(* Logix 5000 project; controller Comas_L4 vendor 1 type 14 code 193 rev 30.11; software revision 30.02; part 2 of 12 *)
(* tags used below, declared in another part *)
   Preposition_OK : BOOL;
(* Engage_Axe, continued *)

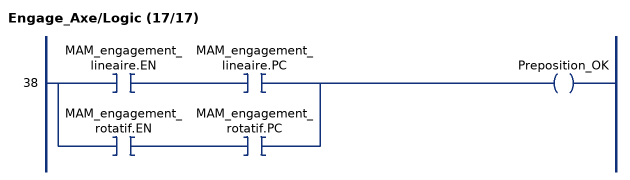
   38: [XIC(MAM_engagement_lineaire.EN) XIC(MAM_engagement_lineaire.PC) ,XIC(MAM_engagement_rotatif.EN) XIC(MAM_engagement_rotatif.PC) ]OTE(Preposition_OK);
END_ROUTINE
END_ADD_ON_INSTRUCTION

ADD_ON_INSTRUCTION Engage_Axe_Virtuel   (* revision 1.11 *)
// Revision note:
// v1.11: Modification Changement de Came en Synchro
// v1.10: Ajout des zones de changement de came
//            Mode Vnul optimisé
// v1.9: Correction Bug maitre à l'arret dans zone d'embrayage: (L16)
//    - Optimisation avec pending status
//    - Forward Only / Bi direc sur MAPC
//    - Command pos au lieu de actual pos sur MAPC
// v1.8: Lancement de came en mode Once (L17)
// v1.7: Degagemennt en position sur front (L8)
// v1.6: Retour cam engage Correct
// v1.5: Ajout modulo esclave
VAR_IN_OUT
   Axe : AXIS_VIRTUAL; {required}   // Axe esclave a controler
   Axe_Maitre : AXIS_VIRTUAL; {required}   // Axe maitre de la came
END_VAR
VAR_INPUT
   Activation : BOOL; {required}   // Activation puissance A Activer avant d'engager
   Engagement : BOOL; {required}   // Engagement de l'axe sur profil de came
   Maitre_V_Nul : BOOL; {required}   // Engagement avec Maitre vitesse nul (positionnement à l'arret)
   Engagement_Decalage : BOOL; {required}   // Activation du decalage en marche
   Degagement_en_pos : BOOL; {required}   // Attente position pour degagement
   Val_Vitesse : REAL; {required}   // Valeur de vitesse global de l'axe
   Val_Acc : REAL; {required}   // Valeur d accel gloable de laxe
   Val_Dec : REAL; {required}   // Valeur de decel
   Val_Jerk : REAL; {required}   // Valeur de jerk
   Val_Engagement : REAL; {required}   // Valeur Absolu d'engagement (0 ou 1 pour axe rotatif)
   Val_Degagement : REAL; {required}   // Valeur de degagement de l'axe (0 ou 1 pour axe rotatif)
   Val_Phase : REAL; {required}   // Valeur de Phase
   Val_Decalage : REAL; {required}   // Valeur de decalage (actif si bit d'activation a 1)
END_VAR
VAR_IN_OUT
   Came : CAM[100]; {required}   // Came modifiable a la volée (tableau de la came)
END_VAR
VAR_INPUT
   Longeur_Cam : DINT; {required}   // Longeur de la came (doit etre sup a 3)
   Modulo_Maitre : REAL; {required}   // Longeur du maitre pour calcul de la phase (modulo maitre)
   Mode_Rotatif : BOOL; {required}   // Activation mode rotatif (MAM type 2 au lieu de 0 pour le pre positionnement)
   Modulo_Esclave : DINT; {required}   // Utilise seulement pour engagement a vnul et rotatif (valeur du modulo de l'axe rotatif)
END_VAR
VAR_OUTPUT
   Axe_Engage : BOOL; {access Read Only, visible}   // Axe engage sur came
   Axe_Degage : BOOL; {access Read Only, visible}   // Axe Degage
   ER : BOOL; {access Read Only, visible}   // Erreur dans le module (retour des blocs fonction)
END_VAR
VAR_INPUT
   Num_Cam_Vnul : DINT;
   ModeCamOnce : BOOL; {required}   // Came en mode once (actif = 1)
   Top_Once : BOOL; {required}   // Top de lancement en mode once
END_VAR
VAR
   MAS_degagement : MOTION_INSTRUCTION;
   MAS_Engagement : MOTION_INSTRUCTION;
   MCCP_1 : MOTION_INSTRUCTION;
   Came_Prof_1 : CAM_PROFILE[20];
   MAPC_1 : MOTION_INSTRUCTION;
   Front : BOOL;
   Val_Phase_Sauve : REAL;
   Val_Phase_Modifie : REAL;
   MAM_Phase : MOTION_INSTRUCTION;
   Engagement_came : BOOL;
   MAM_decalage : MOTION_INSTRUCTION;
   MCCP_2 : MOTION_INSTRUCTION;
   MCCP_First : MOTION_INSTRUCTION;
   MAPC_First : MOTION_INSTRUCTION;
   Came_Prof_2 : CAM_PROFILE[20];
   Came_Prof_First : CAM_PROFILE[20];
   MAPC_2 : MOTION_INSTRUCTION;
   Top_Calage0 : BOOL;
   TEMP_0 : BOOL;
   TEMP_1 : BOOL;
   Top_Calage1 : BOOL;
   Axe_Active : BOOL;
   Num_Cam : DINT;
   Val_phase_modulo : REAL;
   Erreur_1 : BOOL;
   Erreur_2 : BOOL;
   MAS_degagement_enpos : MOTION_INSTRUCTION;
   DEGagement_En_Pos_ok : BOOL;
   Top_Calage2 : BOOL;
   TEMP_2 : BOOL;
   TEMP_3 : BOOL;
   Top_Calage3 : BOOL;
   Val_Engagement_plus : REAL;
   MAM_degagement_rotatif : MOTION_INSTRUCTION;
   MAM_degagement_lineaire : MOTION_INSTRUCTION;
   MAM_degagement_enpos_lineaire : MOTION_INSTRUCTION;
   MAM_degagement_enpos_rotatif : MOTION_INSTRUCTION;
   MAM_engagement_rotatif : MOTION_INSTRUCTION;
   MAM_engagement_lineaire : MOTION_INSTRUCTION;
   Degagement_en_pos_demande : BOOL;
   MAS_degagement_maitreVnul : MOTION_INSTRUCTION;
   Engagement_came_VNul : BOOL;
   MCCP_First_Vnul : MOTION_INSTRUCTION;
   MCSV_Slave_Value : REAL;
   MCSV_Slope_Value : REAL;
   MCSV_SlopeD_Value : REAL;
   MCSV : MOTION_INSTRUCTION;
   MAM_engagement_lineaire_vnul : MOTION_INSTRUCTION;
   MAM_engagement_rotatifvnul : MOTION_INSTRUCTION;
   Val_MAitre : REAL;
   MAPC_First_Vnul : MOTION_INSTRUCTION;
   Front_vnul : BOOL;
   Val_Phase_Modulo2 : REAL;
   MCCP_1_vnul : MOTION_INSTRUCTION;
   Came_Prof_1_vnul : CAM_PROFILE[20];
   MAPC_1_vnul : MOTION_INSTRUCTION;
   MCCP_2_vnul : MOTION_INSTRUCTION;
   Came_Prof_2_vnul : CAM_PROFILE[20];
   MAPC_2_vnul : MOTION_INSTRUCTION;
   TEMP_5 : BOOL;
   Top_Calage5 : BOOL;
   TEMP_6 : BOOL;
   Top_Calage6 : BOOL;
   Erreur_3 : BOOL;
   Erreur_4 : BOOL;
   Front200 : BOOL;
   Cam_Pending : BOOL;
   Tempo_degagement : TIMER;
   decalage_Vnul_Dem : REAL;
   decalage_Vnul_Dem_modulo : REAL;
   front_degagement : BOOL; {access None}
   modulo_div2 : REAL := 1.0; {access None}
   MCCP_First_Once : MOTION_INSTRUCTION; {access None}
   Came_Prof_First_Once : CAM_PROFILE[20]; {access None}
   MAPC_First_Once : MOTION_INSTRUCTION; {access None}
   Front_once : BOOL; {access None}
   Synchro_0 : BOOL; {access None}
   Synchro_1 : BOOL; {access None}
   Val_Engagement_plus_min : REAL; {access None}
   Synchro_vnul_0 : BOOL; {access None}
   Synchro_vnul_1 : BOOL; {access None}
END_VAR

ROUTINE Logic   (* ladder *)
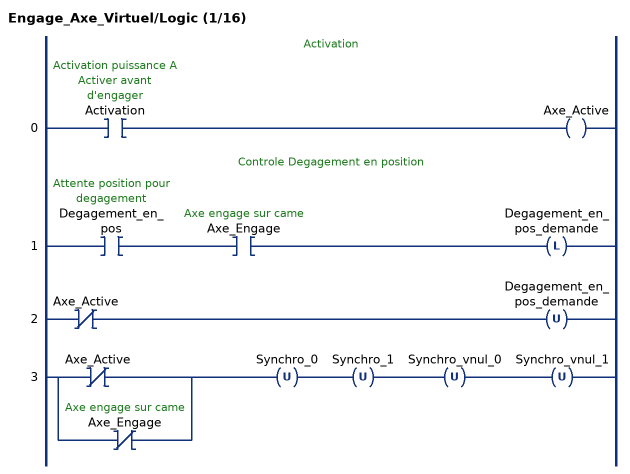
   // Activation
   0: XIC(Activation)OTE(Axe_Active);
   // Controle Degagement en position
   1: XIC(Degagement_en_pos)XIC(Axe_Engage)OTL(Degagement_en_pos_demande);
   2: XIO(Axe_Active)OTU(Degagement_en_pos_demande);
   3: [XIO(Axe_Active) ,XIO(Axe_Engage) ]OTU(Synchro_0)OTU(Synchro_1)OTU(Synchro_vnul_0)OTU(Synchro_vnul_1);
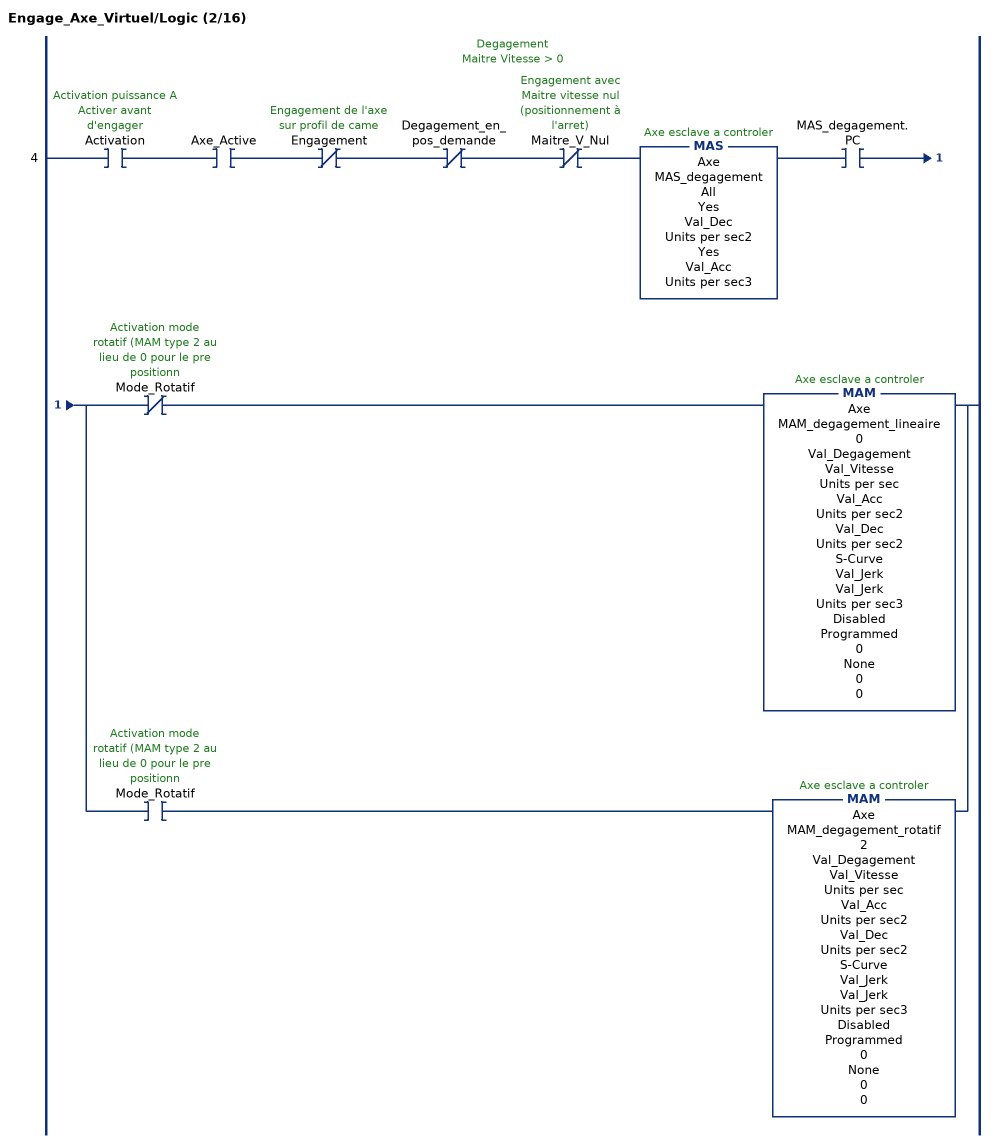
   // Degagement
   // Maitre Vitesse > 0
   4: XIC(Activation)XIC(Axe_Active)XIO(Engagement)XIO(Degagement_en_pos_demande)XIO(Maitre_V_Nul)MAS(Axe,MAS_degagement,All,Yes,Val_Dec,Units per sec2,Yes,Val_Acc,Units per sec3)XIC(MAS_degagement.PC)[XIO(Mode_Rotatif) MAM(Axe,MAM_degagement_lineaire,0,Val_Degagement,Val_Vitesse,Units per sec,Val_Acc,Units per sec2,Val_Dec,Units per sec2,S-Curve,Val_Jerk,Val_Jerk,Units per sec3,Disabled,Programmed,0,None,0,0) ,XIC(Mode_Rotatif) MAM(Axe,MAM_degagement_rotatif,2,Val_Degagement,Val_Vitesse,Units per sec,Val_Acc,Units per sec2,Val_Dec,Units per sec2,S-Curve,Val_Jerk,Val_Jerk,Units per sec3,Disabled,Programmed,0,None,0,0) ];
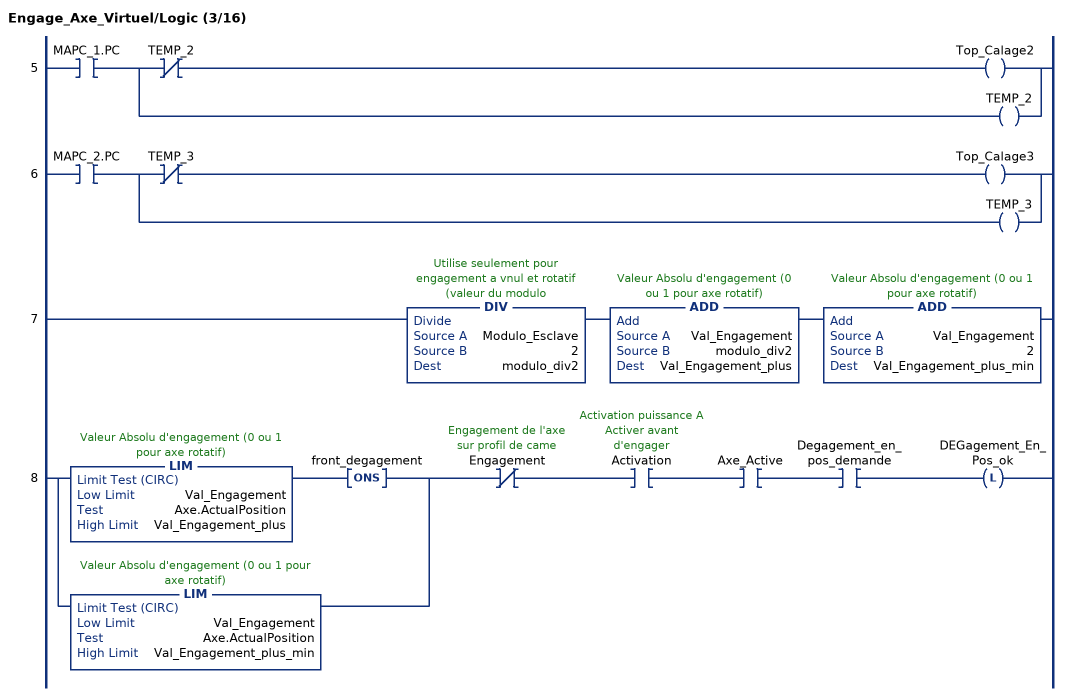
   5: XIC(MAPC_1.PC)[XIO(TEMP_2) OTE(Top_Calage2) ,OTE(TEMP_2) ];
   6: XIC(MAPC_2.PC)[XIO(TEMP_3) OTE(Top_Calage3) ,OTE(TEMP_3) ];
   7: DIV(Modulo_Esclave,2,modulo_div2)ADD(Val_Engagement,modulo_div2,Val_Engagement_plus)ADD(Val_Engagement,2,Val_Engagement_plus_min);
   8: [LIM(Val_Engagement,Axe.ActualPosition,Val_Engagement_plus) ONS(front_degagement) ,LIM(Val_Engagement,Axe.ActualPosition,Val_Engagement_plus_min) ]XIO(Engagement)XIC(Activation)XIC(Axe_Active)XIC(Degagement_en_pos_demande)OTL(DEGagement_En_Pos_ok);
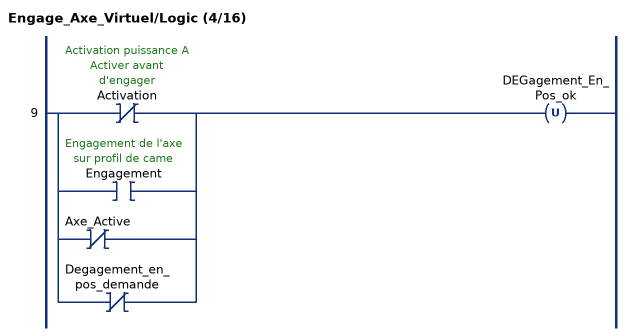
   9: [XIO(Activation) ,XIC(Engagement) ,XIO(Axe_Active) ,XIO(Degagement_en_pos_demande) ]OTU(DEGagement_En_Pos_ok);
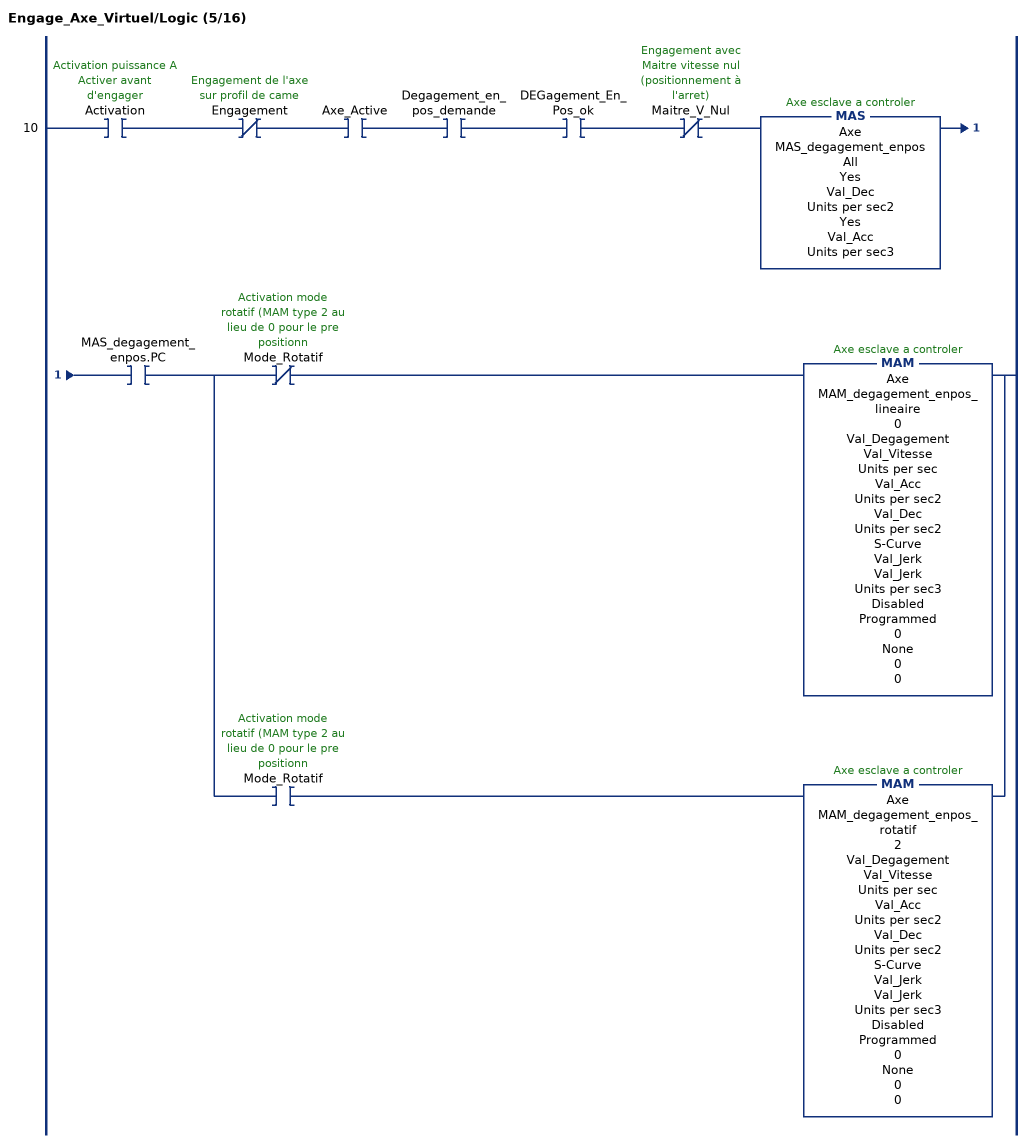
   10: XIC(Activation)XIO(Engagement)XIC(Axe_Active)XIC(Degagement_en_pos_demande)XIC(DEGagement_En_Pos_ok)XIO(Maitre_V_Nul)MAS(Axe,MAS_degagement_enpos,All,Yes,Val_Dec,Units per sec2,Yes,Val_Acc,Units per sec3)XIC(MAS_degagement_enpos.PC)[XIO(Mode_Rotatif) MAM(Axe,MAM_degagement_enpos_lineaire,0,Val_Degagement,Val_Vitesse,Units per sec,Val_Acc,Units per sec2,Val_Dec,Units per sec2,S-Curve,Val_Jerk,Val_Jerk,Units per sec3,Disabled,Programmed,0,None,0,0) ,XIC(Mode_Rotatif) MAM(Axe,MAM_degagement_enpos_rotatif,2,Val_Degagement,Val_Vitesse,Units per sec,Val_Acc,Units per sec2,Val_Dec,Units per sec2,S-Curve,Val_Jerk,Val_Jerk,Units per sec3,Disabled,Programmed,0,None,0,0) ];
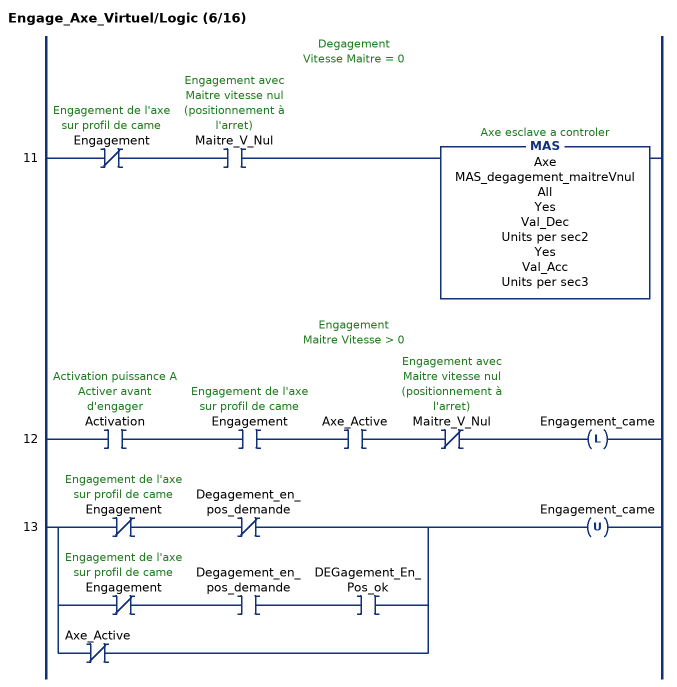
   // Degagement
   // Vitesse Maitre = 0
   11: XIO(Engagement)XIC(Maitre_V_Nul)MAS(Axe,MAS_degagement_maitreVnul,All,Yes,Val_Dec,Units per sec2,Yes,Val_Acc,Units per sec3);
   // Engagement
   // Maitre Vitesse > 0
   12: XIC(Activation)XIC(Engagement)XIC(Axe_Active)XIO(Maitre_V_Nul)OTL(Engagement_came);
   13: [XIO(Engagement) XIO(Degagement_en_pos_demande) ,XIO(Engagement) XIC(Degagement_en_pos_demande) XIC(DEGagement_En_Pos_ok) ,XIO(Axe_Active) ]OTU(Engagement_came);
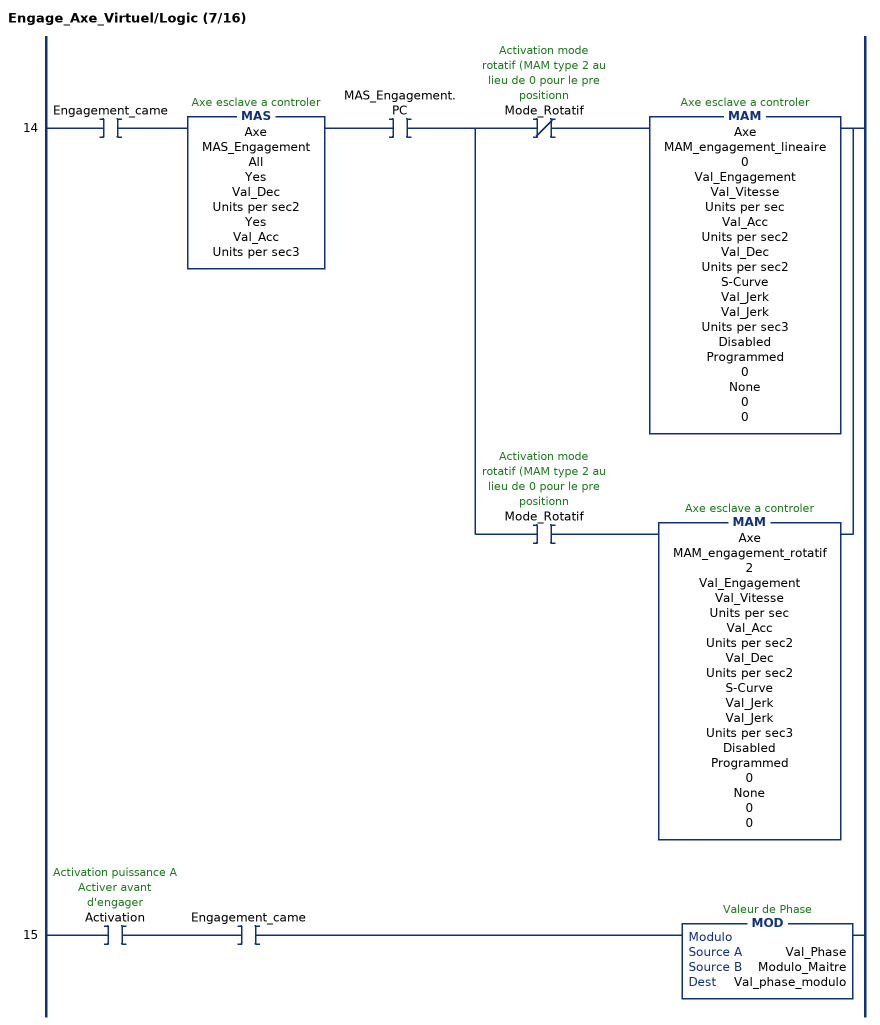
   14: XIC(Engagement_came)MAS(Axe,MAS_Engagement,All,Yes,Val_Dec,Units per sec2,Yes,Val_Acc,Units per sec3)XIC(MAS_Engagement.PC)[XIO(Mode_Rotatif) MAM(Axe,MAM_engagement_lineaire,0,Val_Engagement,Val_Vitesse,Units per sec,Val_Acc,Units per sec2,Val_Dec,Units per sec2,S-Curve,Val_Jerk,Val_Jerk,Units per sec3,Disabled,Programmed,0,None,0,0) ,XIC(Mode_Rotatif) MAM(Axe,MAM_engagement_rotatif,2,Val_Engagement,Val_Vitesse,Units per sec,Val_Acc,Units per sec2,Val_Dec,Units per sec2,S-Curve,Val_Jerk,Val_Jerk,Units per sec3,Disabled,Programmed,0,None,0,0) ];
   15: XIC(Activation)XIC(Engagement_came)MOD(Val_Phase,Modulo_Maitre,Val_phase_modulo);
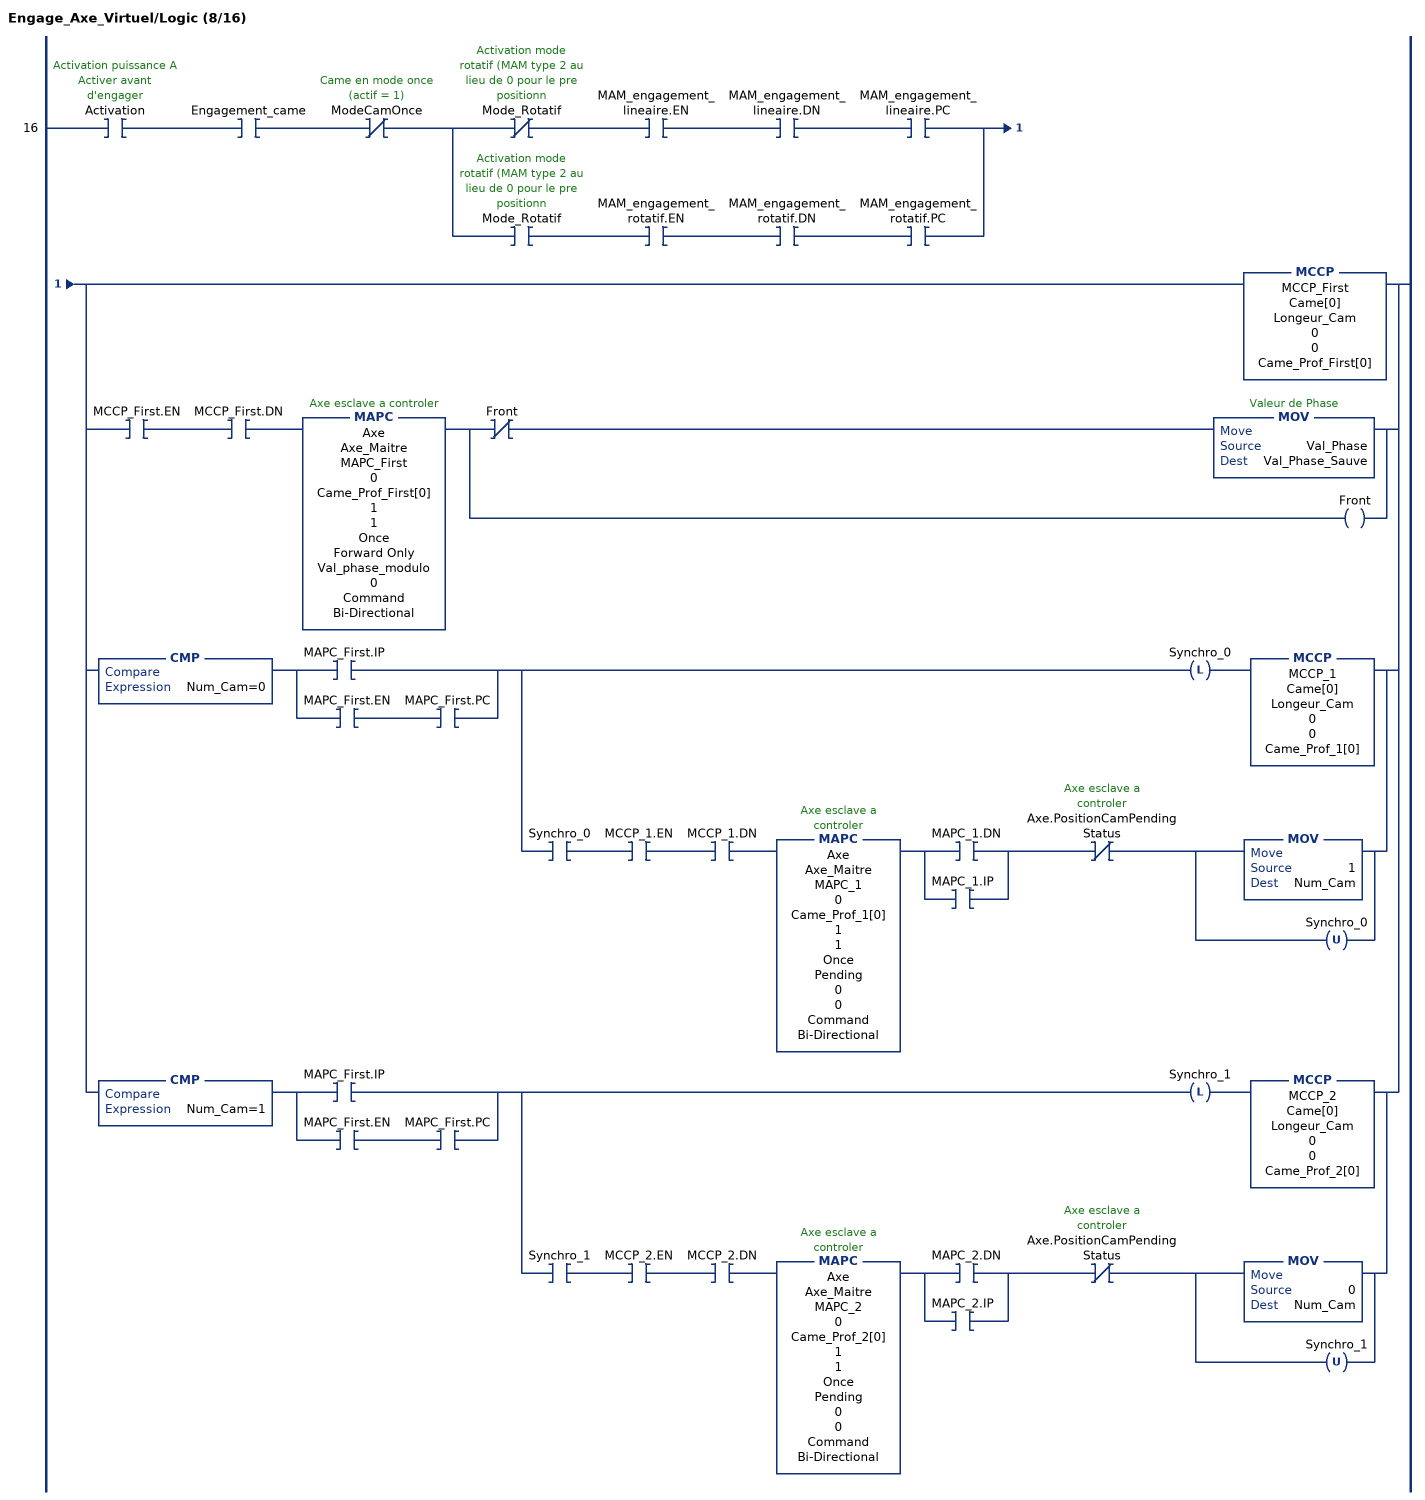
   16: XIC(Activation)XIC(Engagement_came)XIO(ModeCamOnce)[XIO(Mode_Rotatif) XIC(MAM_engagement_lineaire.EN) XIC(MAM_engagement_lineaire.DN) XIC(MAM_engagement_lineaire.PC) ,XIC(Mode_Rotatif) XIC(MAM_engagement_rotatif.EN) XIC(MAM_engagement_rotatif.DN) XIC(MAM_engagement_rotatif.PC) ][MCCP(MCCP_First,Came[0],Longeur_Cam,0,0,Came_Prof_First[0]) ,[XIC(MCCP_First.EN) XIC(MCCP_First.DN) MAPC(Axe,Axe_Maitre,MAPC_First,0,Came_Prof_First[0],1,1,Once,Forward Only,Val_phase_modulo,0,Command,Bi-Directional) [XIO(Front) MOV(Val_Phase,Val_Phase_Sauve) ,OTE(Front) ] ,CMP(Num_Cam=0) [XIC(MAPC_First.IP) ,XIC(MAPC_First.EN) XIC(MAPC_First.PC) ] [OTL(Synchro_0) MCCP(MCCP_1,Came[0],Longeur_Cam,0,0,Came_Prof_1[0]) ,XIC(Synchro_0) XIC(MCCP_1.EN) XIC(MCCP_1.DN) MAPC(Axe,Axe_Maitre,MAPC_1,0,Came_Prof_1[0],1,1,Once,Pending,0,0,Command,Bi-Directional) [XIC(MAPC_1.DN) ,XIC(MAPC_1.IP) ] XIO(Axe.PositionCamPendingStatus) [MOV(1,Num_Cam) ,OTU(Synchro_0) ] ] ,CMP(Num_Cam=1) [XIC(MAPC_First.IP) ,XIC(MAPC_First.EN) XIC(MAPC_First.PC) ] [OTL(Synchro_1) MCCP(MCCP_2,Came[0],Longeur_Cam,0,0,Came_Prof_2[0]) ,XIC(Synchro_1) XIC(MCCP_2.EN) XIC(MCCP_2.DN) MAPC(Axe,Axe_Maitre,MAPC_2,0,Came_Prof_2[0],1,1,Once,Pending,0,0,Command,Bi-Directional) [XIC(MAPC_2.DN) ,XIC(MAPC_2.IP) ] XIO(Axe.PositionCamPendingStatus) [MOV(0,Num_Cam) ,OTU(Synchro_1) ] ] ] ];
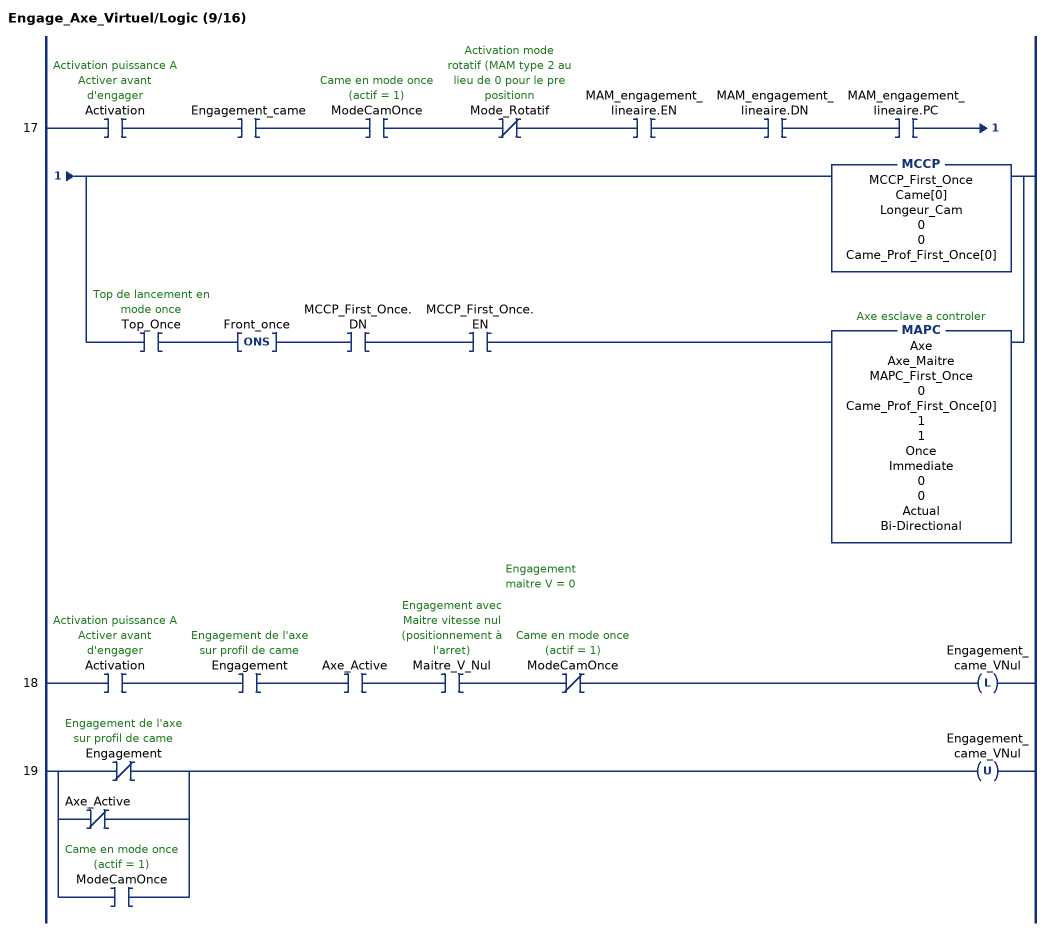
   17: XIC(Activation)XIC(Engagement_came)XIC(ModeCamOnce)XIO(Mode_Rotatif)XIC(MAM_engagement_lineaire.EN)XIC(MAM_engagement_lineaire.DN)XIC(MAM_engagement_lineaire.PC)[MCCP(MCCP_First_Once,Came[0],Longeur_Cam,0,0,Came_Prof_First_Once[0]) ,XIC(Top_Once) ONS(Front_once) XIC(MCCP_First_Once.DN) XIC(MCCP_First_Once.EN) MAPC(Axe,Axe_Maitre,MAPC_First_Once,0,Came_Prof_First_Once[0],1,1,Once,Immediate,0,0,Actual,Bi-Directional) ];
   // Engagement
   // maitre V = 0
   18: XIC(Activation)XIC(Engagement)XIC(Axe_Active)XIC(Maitre_V_Nul)XIO(ModeCamOnce)OTL(Engagement_came_VNul);
   19: [XIO(Engagement) ,XIO(Axe_Active) ,XIC(ModeCamOnce) ]OTU(Engagement_came_VNul);
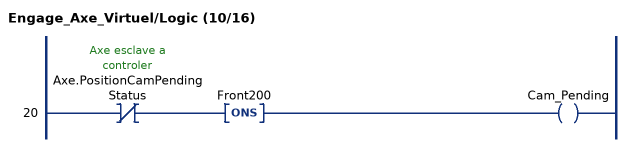
   20: XIO(Axe.PositionCamPendingStatus)ONS(Front200)OTE(Cam_Pending);
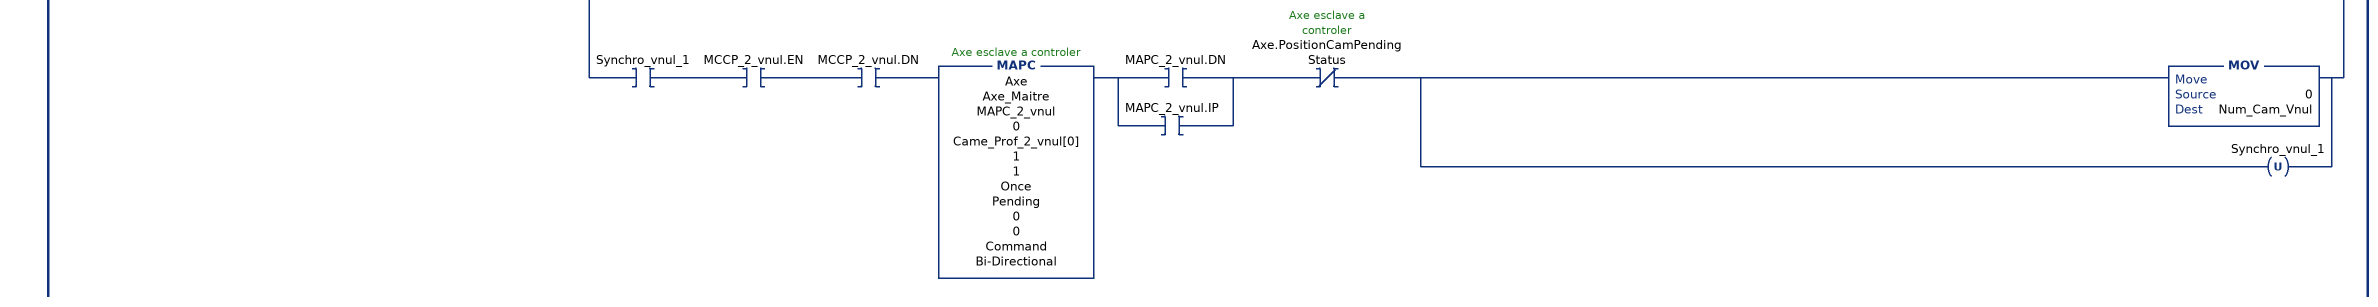
   21: XIC(Engagement_came_VNul)[MCCP(MCCP_First_Vnul,Came[0],Longeur_Cam,0,0,Came_Prof_First[0]) ,XIC(MCCP_First_Vnul.EN) XIC(MCCP_First_Vnul.DN) MOD(Val_Phase,Modulo_Maitre,Val_Phase_Modulo2) SUB(Axe_Maitre.CommandPosition,Val_Phase_Modulo2,Val_MAitre) ADD(Val_MAitre,Modulo_Maitre,Val_MAitre) MOD(Val_MAitre,Modulo_Maitre,Val_MAitre) MCSV(MCSV,Came_Prof_First[0],Val_MAitre,MCSV_Slave_Value,MCSV_Slope_Value,MCSV_SlopeD_Value) ADD(MCSV_Slave_Value,Val_Engagement,decalage_Vnul_Dem) MOD(decalage_Vnul_Dem,Modulo_Esclave,decalage_Vnul_Dem_modulo) XIC(MCSV.DN) [XIO(Mode_Rotatif) MAM(Axe,MAM_engagement_lineaire_vnul,0,decalage_Vnul_Dem,Val_Vitesse,Units per sec,Val_Acc,Units per sec2,Val_Dec,Units per sec2,S-Curve,Val_Jerk,Val_Jerk,Units per sec3,Disabled,Programmed,0,None,0,0) ,XIC(Mode_Rotatif) MAM(Axe,MAM_engagement_rotatifvnul,2,decalage_Vnul_Dem_modulo,Val_Vitesse,Units per sec,Val_Acc,Units per sec2,Val_Dec,Units per sec2,S-Curve,Val_Jerk,Val_Jerk,Units per sec3,Disabled,Programmed,0,None,0,0) ] ,XIC(MCCP_First_Vnul.EN) XIC(MCCP_First_Vnul.DN) MAPC(Axe,Axe_Maitre,MAPC_First_Vnul,0,Came_Prof_First[0],1,1,Once,Immediate,0,Val_MAitre,Command,Bi-Directional) [XIO(Front_vnul) MOV(Val_Phase,Val_Phase_Sauve) ,OTE(Front_vnul) ] ,CMP(Num_Cam_Vnul=0) [XIC(MAPC_First_Vnul.IP) ,XIC(MAPC_First_Vnul.EN) XIC(MAPC_First_Vnul.PC) ] [OTL(Synchro_vnul_0) MCCP(MCCP_1_vnul,Came[0],Longeur_Cam,0,0,Came_Prof_1_vnul[0]) ,XIC(Synchro_vnul_0) XIC(MCCP_1_vnul.EN) XIC(MCCP_1_vnul.DN) MAPC(Axe,Axe_Maitre,MAPC_1_vnul,0,Came_Prof_1_vnul[0],1,1,Once,Pending,0,0,Command,Bi-Directional) [XIC(MAPC_1_vnul.DN) ,XIC(MAPC_1_vnul.IP) ] XIO(Axe.PositionCamPendingStatus) [MOV(1,Num_Cam_Vnul) ,OTU(Synchro_vnul_0) ] ] ,CMP(Num_Cam_Vnul=1) [XIC(MAPC_First_Vnul.IP) ,XIC(MAPC_First_Vnul.EN) XIC(MAPC_First_Vnul.PC) ] [OTL(Synchro_vnul_1) MCCP(MCCP_2_vnul,Came[0],Longeur_Cam,0,0,Came_Prof_2_vnul[0]) ,XIC(Synchro_vnul_1) XIC(MCCP_2_vnul.EN) XIC(MCCP_2_vnul.DN) MAPC(Axe,Axe_Maitre,MAPC_2_vnul,0,Came_Prof_2_vnul[0],1,1,Once,Pending,0,0,Command,Bi-Directional) [XIC(MAPC_2_vnul.DN) ,XIC(MAPC_2_vnul.IP) ] XIO(Axe.PositionCamPendingStatus) [MOV(0,Num_Cam_Vnul) ,OTU(Synchro_vnul_1) ] ] ];
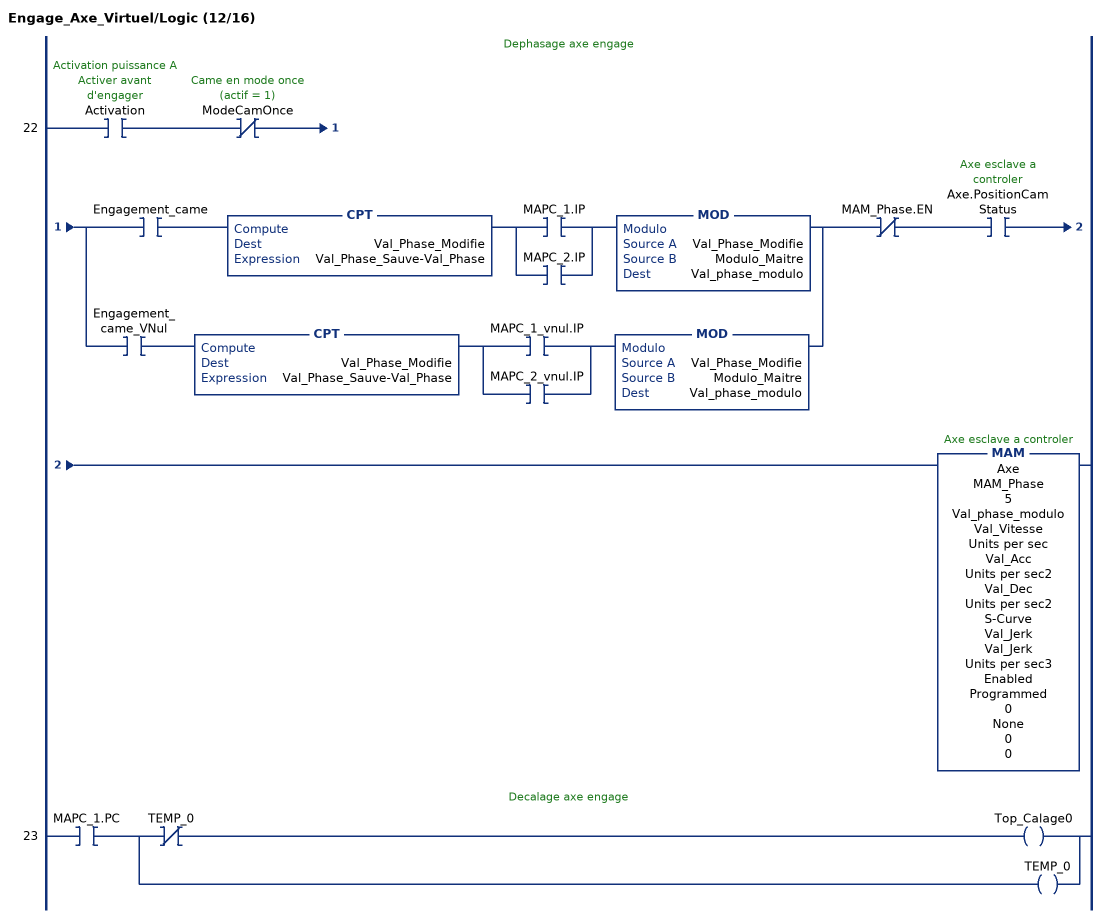
   // Dephasage axe engage
   22: XIC(Activation)XIO(ModeCamOnce)[XIC(Engagement_came) CPT(Val_Phase_Modifie,Val_Phase_Sauve-Val_Phase) [XIC(MAPC_1.IP) ,XIC(MAPC_2.IP) ] MOD(Val_Phase_Modifie,Modulo_Maitre,Val_phase_modulo) ,XIC(Engagement_came_VNul) CPT(Val_Phase_Modifie,Val_Phase_Sauve-Val_Phase) [XIC(MAPC_1_vnul.IP) ,XIC(MAPC_2_vnul.IP) ] MOD(Val_Phase_Modifie,Modulo_Maitre,Val_phase_modulo) ]XIO(MAM_Phase.EN)XIC(Axe.PositionCamStatus)MAM(Axe,MAM_Phase,5,Val_phase_modulo,Val_Vitesse,Units per sec,Val_Acc,Units per sec2,Val_Dec,Units per sec2,S-Curve,Val_Jerk,Val_Jerk,Units per sec3,Enabled,Programmed,0,None,0,0);
   // Decalage axe engage
   23: XIC(MAPC_1.PC)[XIO(TEMP_0) OTE(Top_Calage0) ,OTE(TEMP_0) ];
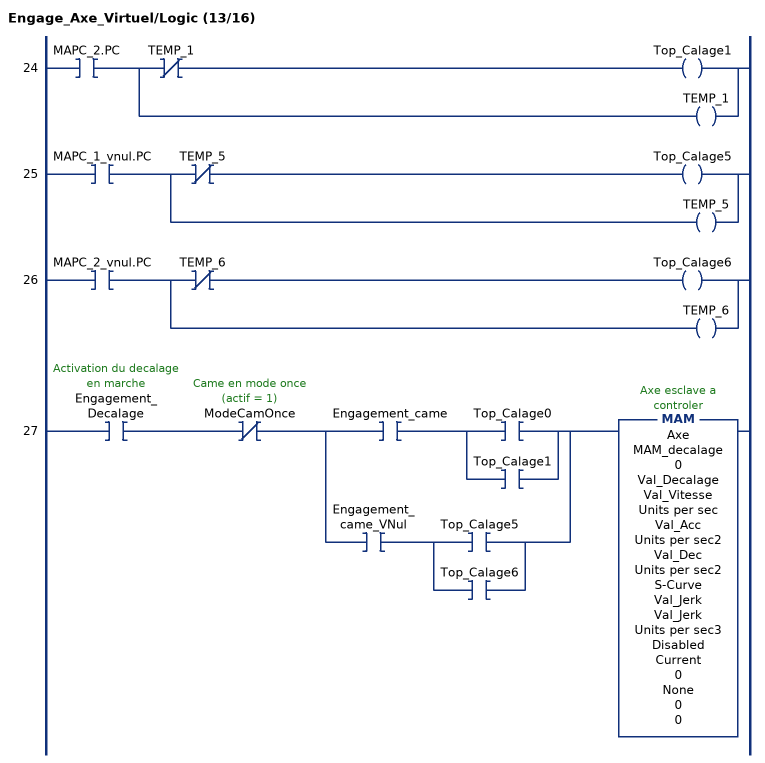
   24: XIC(MAPC_2.PC)[XIO(TEMP_1) OTE(Top_Calage1) ,OTE(TEMP_1) ];
   25: XIC(MAPC_1_vnul.PC)[XIO(TEMP_5) OTE(Top_Calage5) ,OTE(TEMP_5) ];
   26: XIC(MAPC_2_vnul.PC)[XIO(TEMP_6) OTE(Top_Calage6) ,OTE(TEMP_6) ];
   27: XIC(Engagement_Decalage)XIO(ModeCamOnce)[XIC(Engagement_came) [XIC(Top_Calage0) ,XIC(Top_Calage1) ] ,XIC(Engagement_came_VNul) [XIC(Top_Calage5) ,XIC(Top_Calage6) ] ]MAM(Axe,MAM_decalage,0,Val_Decalage,Val_Vitesse,Units per sec,Val_Acc,Units per sec2,Val_Dec,Units per sec2,S-Curve,Val_Jerk,Val_Jerk,Units per sec3,Disabled,Current,0,None,0,0);
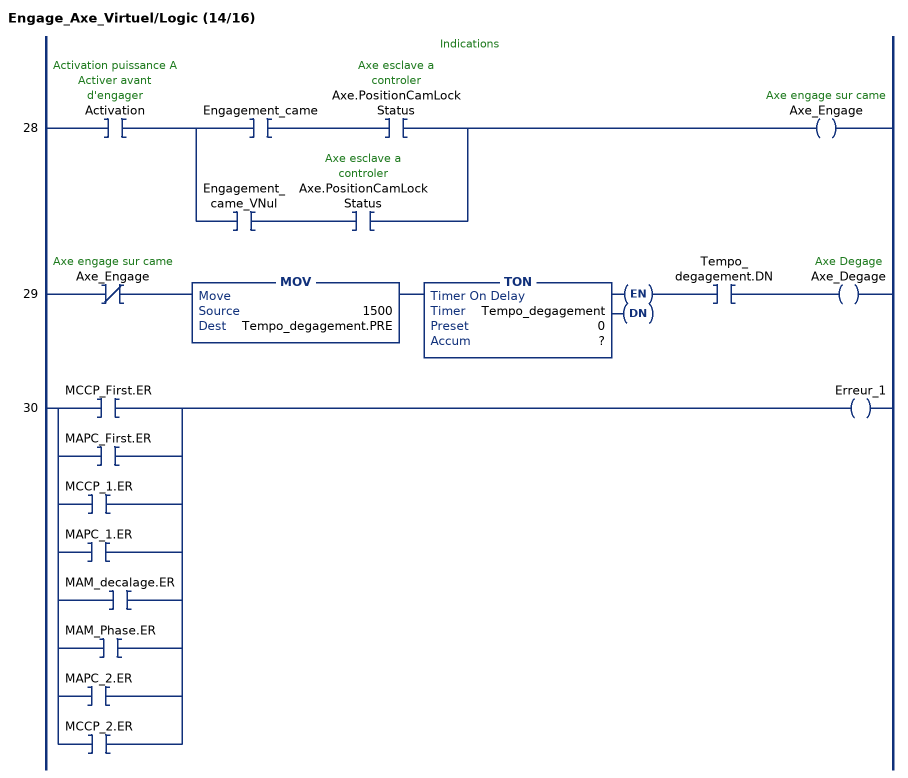
   // Indications
   28: XIC(Activation)[XIC(Engagement_came) XIC(Axe.PositionCamLockStatus) ,XIC(Engagement_came_VNul) XIC(Axe.PositionCamLockStatus) ]OTE(Axe_Engage);
   29: XIO(Axe_Engage)MOV(1500,Tempo_degagement.PRE)TON(Tempo_degagement,?,?)XIC(Tempo_degagement.DN)OTE(Axe_Degage);
   30: [XIC(MCCP_First.ER) ,XIC(MAPC_First.ER) ,XIC(MCCP_1.ER) ,XIC(MAPC_1.ER) ,XIC(MAM_decalage.ER) ,XIC(MAM_Phase.ER) ,XIC(MAPC_2.ER) ,XIC(MCCP_2.ER) ]OTE(Erreur_1);
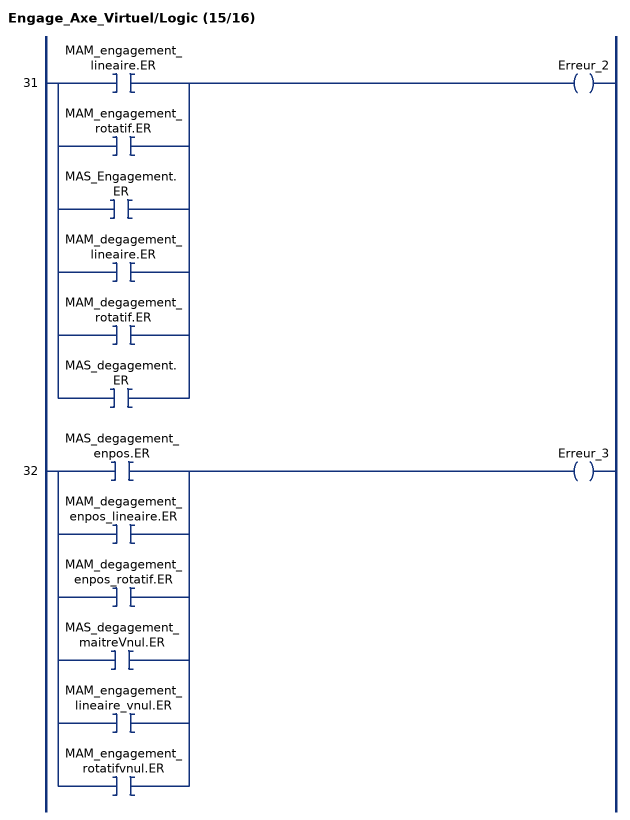
   31: [[XIC(MAM_engagement_lineaire.ER) ,XIC(MAM_engagement_rotatif.ER) ] ,XIC(MAS_Engagement.ER) ,[XIC(MAM_degagement_lineaire.ER) ,XIC(MAM_degagement_rotatif.ER) ] ,XIC(MAS_degagement.ER) ]OTE(Erreur_2);
   32: [XIC(MAS_degagement_enpos.ER) ,[XIC(MAM_degagement_enpos_lineaire.ER) ,[XIC(MAM_degagement_enpos_rotatif.ER) ,[XIC(MAS_degagement_maitreVnul.ER) ,[XIC(MAM_engagement_lineaire_vnul.ER) ,XIC(MAM_engagement_rotatifvnul.ER) ] ] ] ] ]OTE(Erreur_3);
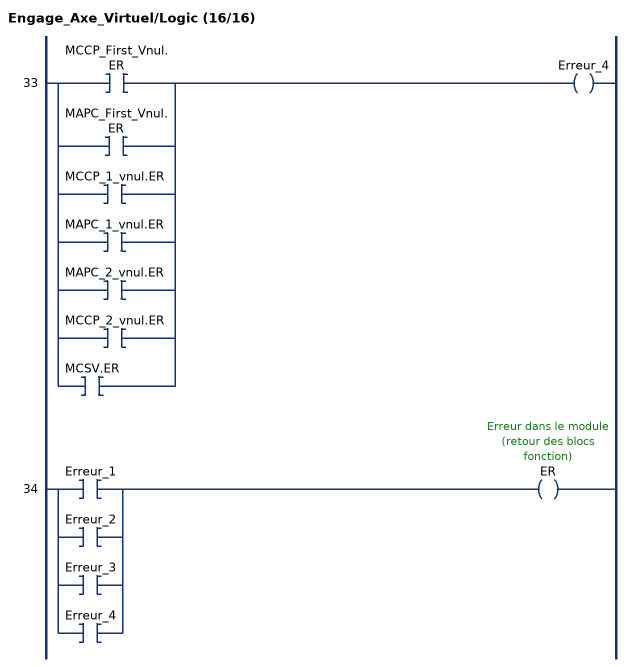
   33: [XIC(MCCP_First_Vnul.ER) ,XIC(MAPC_First_Vnul.ER) ,XIC(MCCP_1_vnul.ER) ,XIC(MAPC_1_vnul.ER) ,XIC(MAPC_2_vnul.ER) ,XIC(MCCP_2_vnul.ER) ,XIC(MCSV.ER) ]OTE(Erreur_4);
   34: [XIC(Erreur_1) ,XIC(Erreur_2) ,XIC(Erreur_3) ,XIC(Erreur_4) ]OTE(ER);
END_ROUTINE
END_ADD_ON_INSTRUCTION

ADD_ON_INSTRUCTION Init_Axe_CIP   (* revision 1.2 *)
// Revision note:
// v1.2 correction arret axe
VAR_IN_OUT
   Axe : AXIS_CIP_DRIVE; {required}
END_VAR
VAR_INPUT
   Init : BOOL; {required}   // Lancement sequence init
   Direction_Capteur : BOOL; {required}   // 0= sens positif
   Sens_Capteur : BOOL; {required}   // 0 = front montant
   Vitesse : REAL; {required}
   Acc : REAL; {required}
   Dec : REAL; {required}
   Jerk : REAL; {required}
END_VAR
VAR_OUTPUT
   IP : BOOL; {access Read Only, visible}
   ER : BOOL; {access Read Only, visible}
   Init_OK : BOOL; {access Read Only, visible}
END_VAR
VAR
   MAJ_Test : MOTION_INSTRUCTION;
   MSO_Test : MOTION_INSTRUCTION;
   Temp : BOOL;
   MSF_Test : MOTION_INSTRUCTION;
   MSO_Test_Positif : MOTION_INSTRUCTION;
   MSO_Test_negatif : MOTION_INSTRUCTION;
   MAJ_Test_Positif : MOTION_INSTRUCTION;
   MAJ_Test_Negatif : MOTION_INSTRUCTION;
   MASR_AXE : MOTION_INSTRUCTION;
   MAFR_AXE : MOTION_INSTRUCTION;
   MAS_AXE : MOTION_INSTRUCTION;
   TON_Test : TIMER;
   MCD_Jog : MOTION_INSTRUCTION;
   erreur_1 : BOOL;
   erreur_2 : BOOL;
   MAH_Axe : MOTION_INSTRUCTION;
   Vitesse_Sens : REAL;
   MAS2_AXE : MOTION_INSTRUCTION;
   temp2 : BOOL;
   TEMP10 : BOOL;
   MASMAH2_AXE : MOTION_INSTRUCTION;
   FRONTCPT : BOOL;
   INITENCOURS : BOOL;
   MSF_Test_INIT : MOTION_INSTRUCTION;
   MSO_Test_INIT : MOTION_INSTRUCTION;
   Autorisation : BOOL;
   FRONTCPT2 : BOOL;
   Temp3 : BOOL;
   Temp4 : BOOL;
   Front_init : BOOL; {access None}
   MAS_Test_Positif : MOTION_INSTRUCTION; {access None}
   MAS_Test_Negatif : MOTION_INSTRUCTION; {access None}
   Axe_Pret_a_bouger : BOOL; {access None}
   MAS_Test_Positif_inv : MOTION_INSTRUCTION; {access None}
   MAJ_Test_Positif_inv : MOTION_INSTRUCTION; {access None}
   MAS_Test_Negatif_inv : MOTION_INSTRUCTION; {access None}
   MAJ_Test_Negatif_inv : MOTION_INSTRUCTION; {access None}
   Init_ONS : BOOL; {access None}
   Etape_Init : DINT; {access None}
   FRONTCPT3 : BOOL; {access None}
   FRONTCPT4 : BOOL; {access None}
   Init_ONS_off : BOOL; {access None}
   front_init_off : BOOL; {access None}
   MSF_Test_INIT_off : MOTION_INSTRUCTION; {access None}
   not_ip : BOOL; {access None}
   Tempo_MAH : TIMER; {access None}
   MAS_arret_init : MOTION_INSTRUCTION; {access None}
   Tempo_Msf : TIMER; {access None}
END_VAR

ROUTINE Logic   (* ladder *)
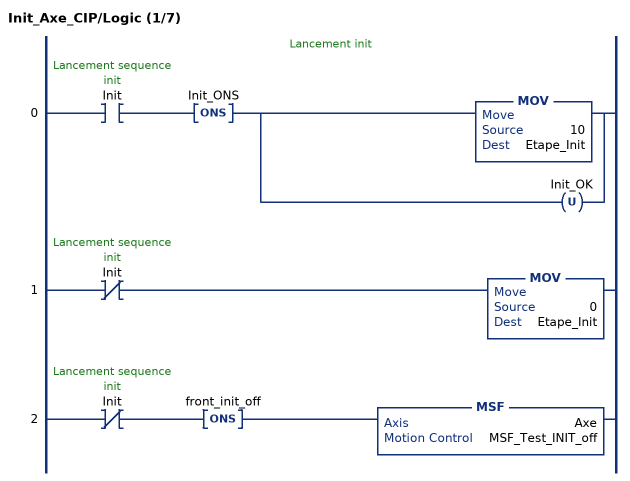
   // Lancement init
   0: XIC(Init)ONS(Init_ONS)[MOV(10,Etape_Init) ,OTU(Init_OK) ];
   1: XIO(Init)MOV(0,Etape_Init);
   2: XIO(Init)ONS(front_init_off)MSF(Axe,MSF_Test_INIT_off);
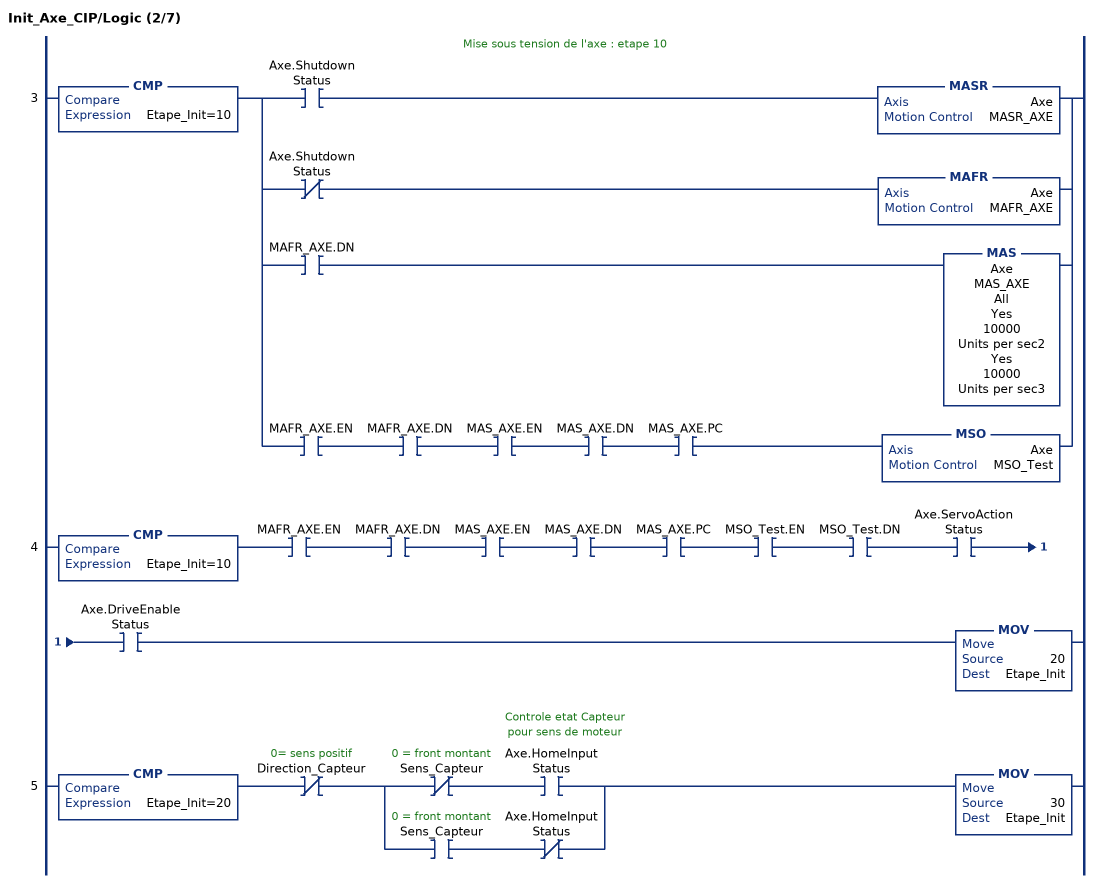
   // Mise sous tension de l'axe : etape 10
   3: CMP(Etape_Init=10)[[XIC(Axe.ShutdownStatus) MASR(Axe,MASR_AXE) ,XIO(Axe.ShutdownStatus) MAFR(Axe,MAFR_AXE) ,XIC(MAFR_AXE.DN) MAS(Axe,MAS_AXE,All,Yes,10000,Units per sec2,Yes,10000,Units per sec3) ] ,XIC(MAFR_AXE.EN) XIC(MAFR_AXE.DN) XIC(MAS_AXE.EN) XIC(MAS_AXE.DN) XIC(MAS_AXE.PC) MSO(Axe,MSO_Test) ];
   4: CMP(Etape_Init=10)XIC(MAFR_AXE.EN)XIC(MAFR_AXE.DN)XIC(MAS_AXE.EN)XIC(MAS_AXE.DN)XIC(MAS_AXE.PC)XIC(MSO_Test.EN)XIC(MSO_Test.DN)XIC(Axe.ServoActionStatus)XIC(Axe.DriveEnableStatus)MOV(20,Etape_Init);
   // Controle etat Capteur
   // pour sens de moteur
   5: CMP(Etape_Init=20)XIO(Direction_Capteur)[XIO(Sens_Capteur) XIC(Axe.HomeInputStatus) ,XIC(Sens_Capteur) XIO(Axe.HomeInputStatus) ]MOV(30,Etape_Init);
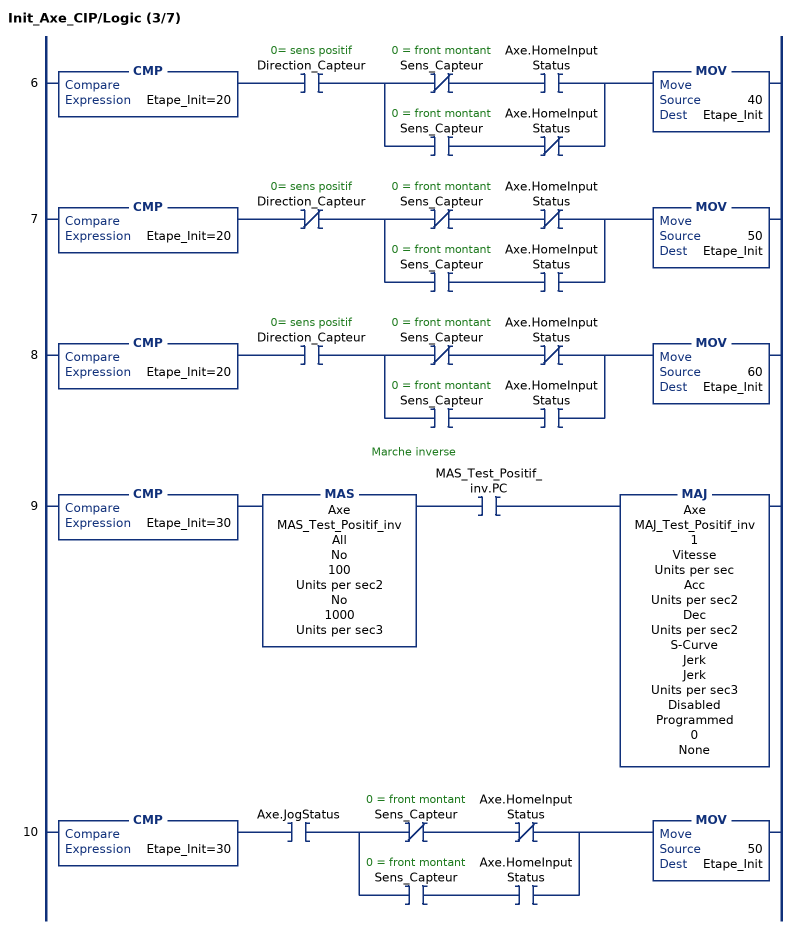
   6: CMP(Etape_Init=20)XIC(Direction_Capteur)[XIO(Sens_Capteur) XIC(Axe.HomeInputStatus) ,XIC(Sens_Capteur) XIO(Axe.HomeInputStatus) ]MOV(40,Etape_Init);
   7: CMP(Etape_Init=20)XIO(Direction_Capteur)[XIO(Sens_Capteur) XIO(Axe.HomeInputStatus) ,XIC(Sens_Capteur) XIC(Axe.HomeInputStatus) ]MOV(50,Etape_Init);
   8: CMP(Etape_Init=20)XIC(Direction_Capteur)[XIO(Sens_Capteur) XIO(Axe.HomeInputStatus) ,XIC(Sens_Capteur) XIC(Axe.HomeInputStatus) ]MOV(60,Etape_Init);
   // Marche inverse
   9: CMP(Etape_Init=30)MAS(Axe,MAS_Test_Positif_inv,All,No,100,Units per sec2,No,1000,Units per sec3)XIC(MAS_Test_Positif_inv.PC)MAJ(Axe,MAJ_Test_Positif_inv,1,Vitesse,Units per sec,Acc,Units per sec2,Dec,Units per sec2,S-Curve,Jerk,Jerk,Units per sec3,Disabled,Programmed,0,None);
   10: CMP(Etape_Init=30)XIC(Axe.JogStatus)[XIO(Sens_Capteur) XIO(Axe.HomeInputStatus) ,XIC(Sens_Capteur) XIC(Axe.HomeInputStatus) ]MOV(50,Etape_Init);
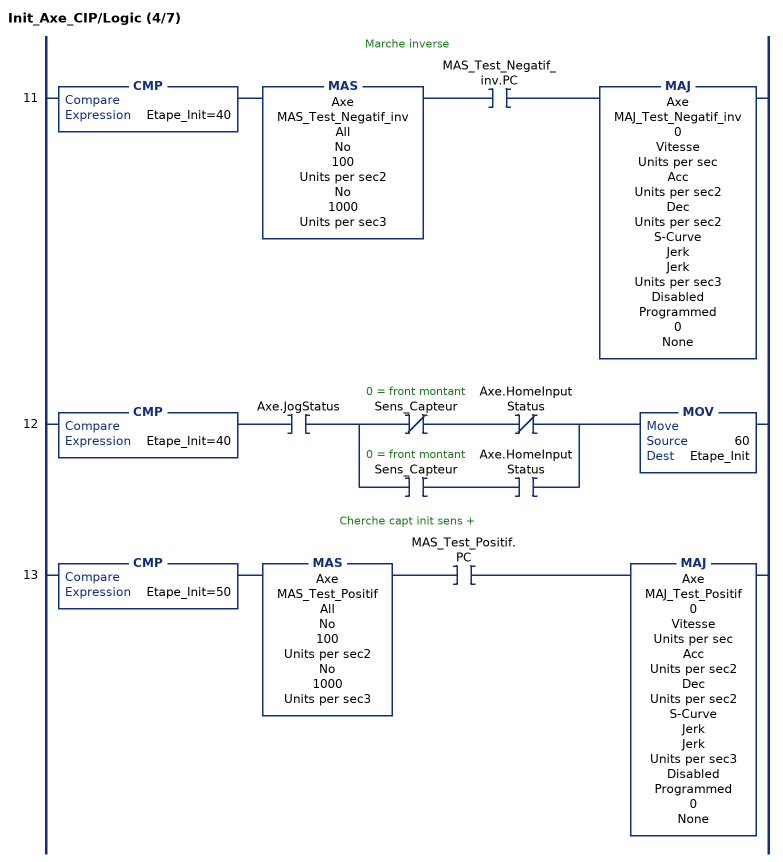
   // Marche inverse
   11: CMP(Etape_Init=40)MAS(Axe,MAS_Test_Negatif_inv,All,No,100,Units per sec2,No,1000,Units per sec3)XIC(MAS_Test_Negatif_inv.PC)MAJ(Axe,MAJ_Test_Negatif_inv,0,Vitesse,Units per sec,Acc,Units per sec2,Dec,Units per sec2,S-Curve,Jerk,Jerk,Units per sec3,Disabled,Programmed,0,None);
   12: CMP(Etape_Init=40)XIC(Axe.JogStatus)[XIO(Sens_Capteur) XIO(Axe.HomeInputStatus) ,XIC(Sens_Capteur) XIC(Axe.HomeInputStatus) ]MOV(60,Etape_Init);
   // Cherche capt init sens +
   13: CMP(Etape_Init=50)MAS(Axe,MAS_Test_Positif,All,No,100,Units per sec2,No,1000,Units per sec3)XIC(MAS_Test_Positif.PC)MAJ(Axe,MAJ_Test_Positif,0,Vitesse,Units per sec,Acc,Units per sec2,Dec,Units per sec2,S-Curve,Jerk,Jerk,Units per sec3,Disabled,Programmed,0,None);
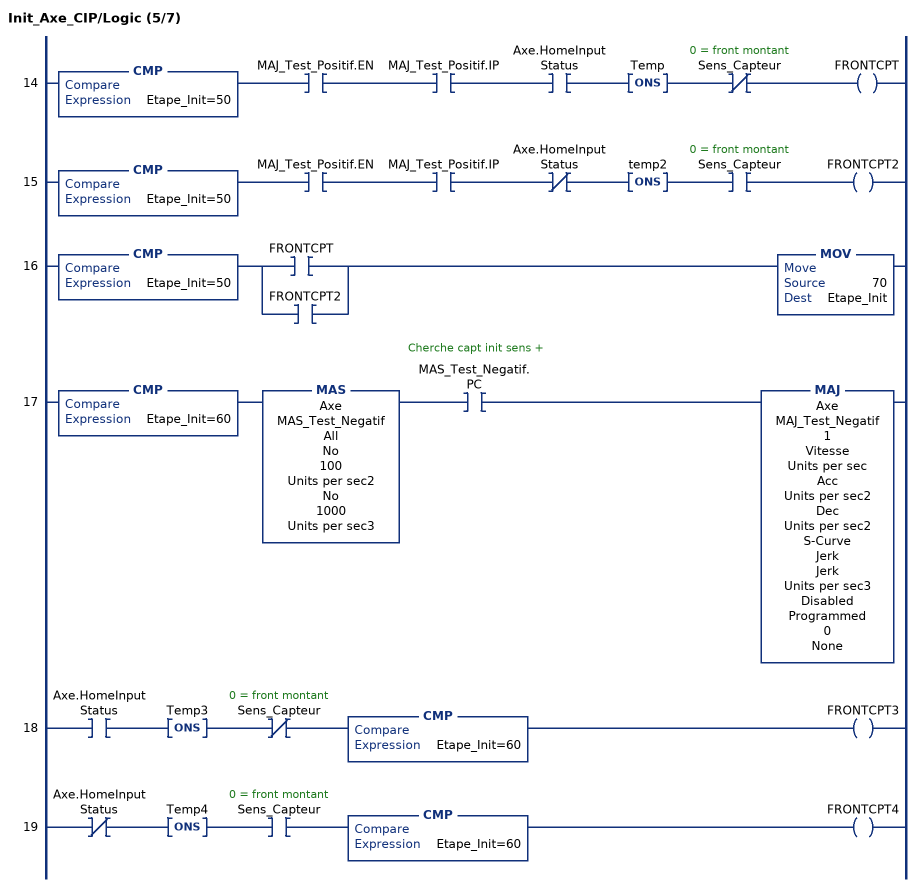
   14: CMP(Etape_Init=50)XIC(MAJ_Test_Positif.EN)XIC(MAJ_Test_Positif.IP)XIC(Axe.HomeInputStatus)ONS(Temp)XIO(Sens_Capteur)OTE(FRONTCPT);
   15: CMP(Etape_Init=50)XIC(MAJ_Test_Positif.EN)XIC(MAJ_Test_Positif.IP)XIO(Axe.HomeInputStatus)ONS(temp2)XIC(Sens_Capteur)OTE(FRONTCPT2);
   16: CMP(Etape_Init=50)[XIC(FRONTCPT) ,XIC(FRONTCPT2) ]MOV(70,Etape_Init);
   // Cherche capt init sens +
   17: CMP(Etape_Init=60)MAS(Axe,MAS_Test_Negatif,All,No,100,Units per sec2,No,1000,Units per sec3)XIC(MAS_Test_Negatif.PC)MAJ(Axe,MAJ_Test_Negatif,1,Vitesse,Units per sec,Acc,Units per sec2,Dec,Units per sec2,S-Curve,Jerk,Jerk,Units per sec3,Disabled,Programmed,0,None);
   18: XIC(Axe.HomeInputStatus)ONS(Temp3)XIO(Sens_Capteur)CMP(Etape_Init=60)OTE(FRONTCPT3);
   19: XIO(Axe.HomeInputStatus)ONS(Temp4)XIC(Sens_Capteur)CMP(Etape_Init=60)OTE(FRONTCPT4);
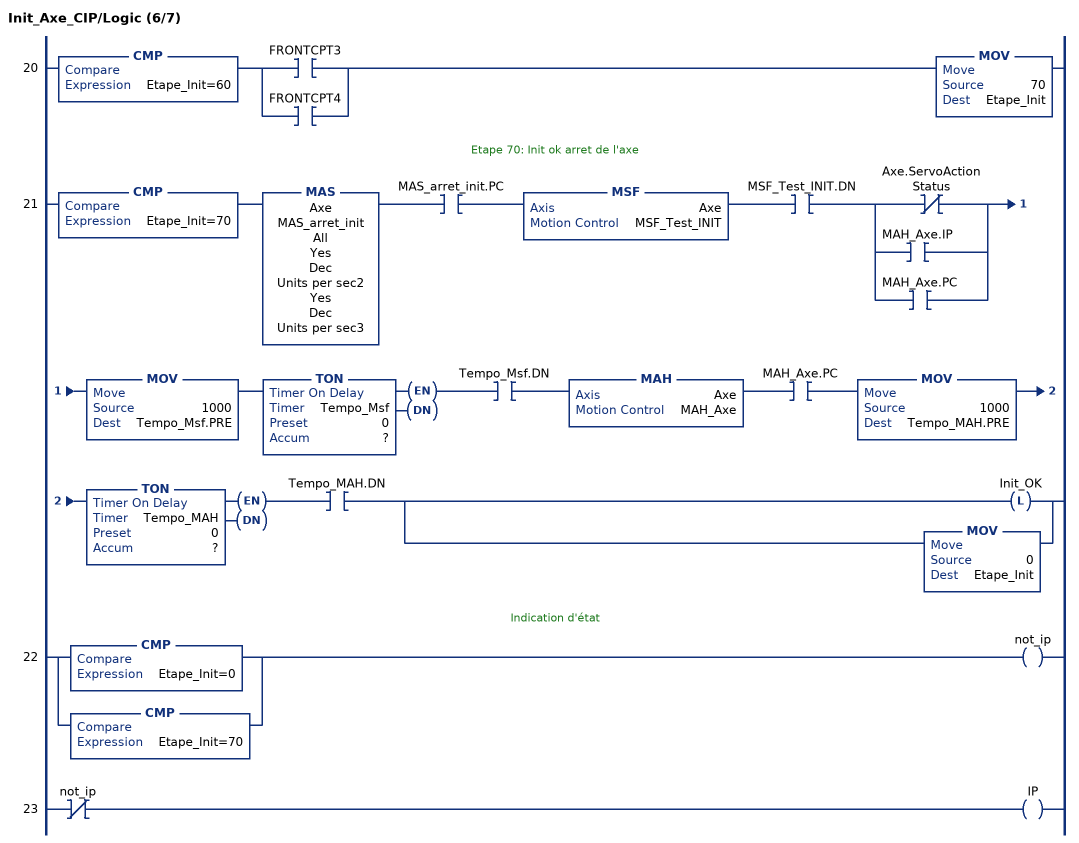
   20: CMP(Etape_Init=60)[XIC(FRONTCPT3) ,XIC(FRONTCPT4) ]MOV(70,Etape_Init);
   // Etape 70: Init ok arret de l'axe
   21: CMP(Etape_Init=70)MAS(Axe,MAS_arret_init,All,Yes,Dec,Units per sec2,Yes,Dec,Units per sec3)XIC(MAS_arret_init.PC)MSF(Axe,MSF_Test_INIT)XIC(MSF_Test_INIT.DN)[XIO(Axe.ServoActionStatus) ,XIC(MAH_Axe.IP) ,XIC(MAH_Axe.PC) ]MOV(1000,Tempo_Msf.PRE)TON(Tempo_Msf,?,?)XIC(Tempo_Msf.DN)MAH(Axe,MAH_Axe)XIC(MAH_Axe.PC)MOV(1000,Tempo_MAH.PRE)TON(Tempo_MAH,?,?)XIC(Tempo_MAH.DN)[OTL(Init_OK) ,MOV(0,Etape_Init) ];
   // Indication d'état
   22: [CMP(Etape_Init=0) ,CMP(Etape_Init=70) ]OTE(not_ip);
   23: XIO(not_ip)OTE(IP);
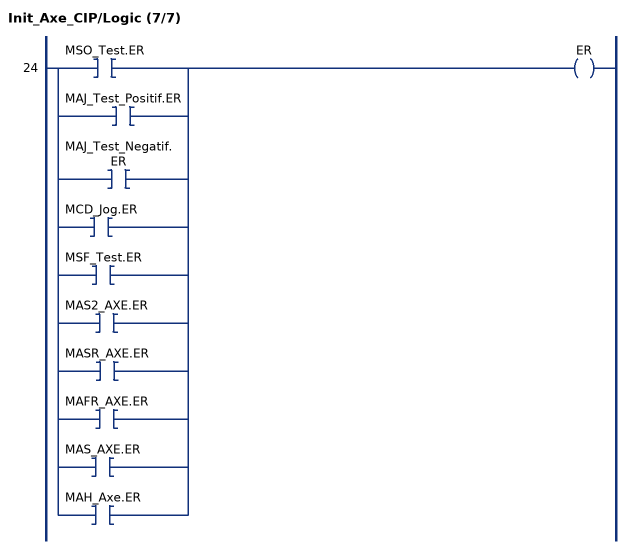
   24: [XIC(MSO_Test.ER) ,[XIC(MAJ_Test_Positif.ER) ,[XIC(MAJ_Test_Negatif.ER) ,[XIC(MCD_Jog.ER) ,[XIC(MSF_Test.ER) ,XIC(MAS2_AXE.ER) ,XIC(MASR_AXE.ER) ,XIC(MAFR_AXE.ER) ,XIC(MAS_AXE.ER) ,XIC(MAH_Axe.ER) ] ] ] ] ]OTE(ER);
END_ROUTINE
END_ADD_ON_INSTRUCTION
